Fanuc KAREL source: kc00031.KL

-- PROVISIONAL review KL for V940-1; original PC SHA256 6b3a1c43933e2a53e173fd1cc13a4a655e4a1b53868524e6112bad552a43931a
-- Incomplete behavior may be omitted. Consult companion uncertainty JSON. Do not deploy.
PROGRAM KC00031
%NOLOCKGROUP
BEGIN
  -- V9_ZERO_TABLE_METADATA_HINT layout=0002_ascii; no indexed target words; source/name/runtime held
  -- UNRESOLVED_PC offsets 5-27; opcodes 27,22,22,31,23
  -- UNRESOLVED_PC offsets 32-36; opcodes 7F
END KC00031
